(* IEC 61131-3 sources: plc_simulator/services/codesys/POUs (part 3) *)

(* ---- FC_TSK_Resolve.st ---- *)
(* ===========================================================================================
 *  FC_TSK_Resolve — Conflict resolution
 *
 *  Company : Galvatek part of the John Cockerill Group
 *  Author  : Jarmo Piipponen
 *  Created : 25.03.2026
 *
 * -------------------------------------------------------------------------------------------
 *  Four sequential resolution phases:
 *  1. ADVANCE (chain bottleneck + suffix flex_down)
 *  2. DELAY (single-stage vFlexUp)
 *  3. PRECEDING_DELAY (conf stage-1)
 *  4. DELAY_PREV_PAST_NEXT (force order swap)
 *
 *  VAR_IN_OUT: ioSchedule, ioTask, ioBatch, ioLocks,
 *  ioLockCnt — caller passes live or workspace arrays.
 *
 *  ------------------------------------------------------------------------------------------
 *
 *  Changes:
 *
 *
 *
 *)

FUNCTION FC_TSK_Resolve : BOOL

(* Introduction of Variables ----------------------------------------------------------------*)

VAR_INPUT
  iConfUnit               : INT;
  iConfStage              : INT;
  iConfTrans              : INT;
  iBlockedUnit            : INT;
  iBlockedStage           : INT;
  iDeficit                 : REAL;
END_VAR

VAR_IN_OUT  (* array sizes must match GVL_JC_Constants: 50=MAX_LOCKS, 10=MAX_UNITS, 3=MAX_TRANSPORTERS *)
  ioLocks                  : ARRAY[1..50] OF UDT_JC_TskLockType;
  ioLockCnt               : INT;
  ioSchedule               : ARRAY[1..10] OF UDT_JC_TskScheduleType;
  ioTask                   : ARRAY[1..3] OF UDT_JC_TskQueueType;
  ioBatch                  : ARRAY[1..10] OF UDT_BatchType;
END_VAR

VAR_EXTERNAL CONSTANT
    MAX_TRANSPORTERS        : INT;
    MAX_UNITS               : INT;
    SCH_TSK_FLEX_FACTOR     : REAL;
END_VAR

VAR_OUTPUT
  oSolved                  : BOOL;
  oTotalDelay             : REAL;
  oTotalAdv               : REAL;
END_VAR

VAR
  vRemain                    : REAL;
  cap                       : REAL;
  vAmount                    : REAL;
  vStageFlex                : REAL;
  is_locked_adv             : BOOL;
  is_locked_del             : BOOL;
  vCanAdvance               : BOOL;
  vCanDelay                 : BOOL;
  vLockI                    : INT;
  vPrevConfStage           : INT;
  is_pcs_locked             : BOOL;
  vPrevSinkStn             : INT;
  vNextLiftStn             : INT;
  is_blk_adv_locked         : BOOL;
  qi                        : INT;
  vChainFlex                : REAL;
  vSuffixFlex               : REAL;
  earlier_stg               : INT;
  earlier_flex              : REAL;
  vChainAmount              : REAL;
  vSuffixAmount             : REAL;
  vSchedBlocked             : INT;
  vSchedConf                : INT;
  vSchedPrevConf           : INT;
  vTmpSi                    : INT;
  cap_remain                : REAL;
END_VAR

FC_TSK_Resolve := FALSE;
oSolved      := FALSE;
oTotalDelay := 0.0;
oTotalAdv   := 0.0;
vRemain        := iDeficit;

IF vRemain <= 0.1 THEN
  oSolved := TRUE;
  FC_TSK_Resolve := TRUE;
  RETURN;
END_IF;

(* Lock check: blocked stage locked DELAY? cannot ADVANCE *)
is_locked_adv := FALSE;
FOR vLockI := 1 TO ioLockCnt DO
  IF ioLocks[vLockI].Unit = iBlockedUnit
     AND ioLocks[vLockI].Stage = iBlockedStage
     AND ioLocks[vLockI].Direction = 2 THEN
    is_locked_adv := TRUE;
  END_IF;
END_FOR;

(* Lock check: conf stage locked ADVANCE? cannot DELAY *)
is_locked_del := FALSE;
FOR vLockI := 1 TO ioLockCnt DO
  IF ioLocks[vLockI].Unit = iConfUnit
     AND ioLocks[vLockI].Stage = iConfStage
     AND ioLocks[vLockI].Direction = 1 THEN
    is_locked_del := TRUE;
  END_IF;
END_FOR;

vCanAdvance := NOT is_locked_adv;
vCanDelay   := NOT is_locked_del;

(* Map ProgramStage to schedule array index *)
vSchedBlocked := 0;
IF iBlockedUnit >= 1 AND iBlockedUnit <= MAX_UNITS THEN
  FOR vTmpSi := 1 TO ioSchedule[iBlockedUnit].StageCount DO
    IF ioSchedule[iBlockedUnit].Stages[vTmpSi].ProgramStage = iBlockedStage THEN
      vSchedBlocked := vTmpSi; EXIT;
    END_IF;
  END_FOR;
END_IF;

vSchedConf := 0;
IF iConfUnit >= 1 AND iConfUnit <= MAX_UNITS THEN
  FOR vTmpSi := 1 TO ioSchedule[iConfUnit].StageCount DO
    IF ioSchedule[iConfUnit].Stages[vTmpSi].ProgramStage = iConfStage THEN
      vSchedConf := vTmpSi; EXIT;
    END_IF;
  END_FOR;
END_IF;

(* ================================================================ *)
(* PHASE 1: ADVANCE -- advance blocked batch                       *)
(* ================================================================ *)
IF vCanAdvance
   AND iBlockedUnit >= 1 AND iBlockedUnit <= MAX_UNITS
   AND iBlockedStage >= 1 THEN
IF vSchedBlocked >= 1 AND vSchedBlocked <= ioSchedule[iBlockedUnit].StageCount THEN

  (* Absolute flex cap: use (MaxTime - MinTime) range, not (CalcTime - MinTime).
     This prevents cumulative drift when CalcTime is vAdjusted across rounds. *)
  vStageFlex := DINT_TO_REAL(
    ioSchedule[iBlockedUnit].Stages[vSchedBlocked].MaxTime
    - ioSchedule[iBlockedUnit].Stages[vSchedBlocked].MinTime);
  IF vStageFlex < 0.0 THEN vStageFlex := 0.0; END_IF;
  vStageFlex := vStageFlex * SCH_TSK_FLEX_FACTOR;
  (* Cap to actual remaining advance room *)
  cap_remain := DINT_TO_REAL(
    ioSchedule[iBlockedUnit].Stages[vSchedBlocked].CalcTime
    - ioSchedule[iBlockedUnit].Stages[vSchedBlocked].MinTime);
  IF cap_remain < 0.0 THEN cap_remain := 0.0; END_IF;
  IF vStageFlex > cap_remain THEN vStageFlex := cap_remain; END_IF;

  IF vStageFlex > 0.1 THEN
    IF ioBatch[iBlockedUnit].CurStage = iBlockedStage THEN cap := 0.9;
  ELSE cap := 0.5; END_IF;

    (* Chain bottleneck search *)
    vChainFlex := vStageFlex;
    FOR earlier_stg := 1 TO vSchedBlocked - 1 DO
      earlier_flex := DINT_TO_REAL(
        ioSchedule[iBlockedUnit].Stages[earlier_stg].CalcTime
        - ioSchedule[iBlockedUnit].Stages[earlier_stg].MinTime);
  IF earlier_flex < 0.0 THEN earlier_flex := 0.0; END_IF;
      IF earlier_flex > 0.0 AND earlier_flex < vChainFlex THEN
        vChainFlex := earlier_flex;
      END_IF;
    END_FOR;

    (* CHAIN_ADVANCE *)
    vChainAmount := vChainFlex * cap;
  IF vChainAmount > vRemain THEN vChainAmount := vRemain; END_IF;

    IF vChainAmount > 0.1 THEN
      ioSchedule[iBlockedUnit].Stages[vSchedBlocked].CalcTime :=
        ioSchedule[iBlockedUnit].Stages[vSchedBlocked].CalcTime - REAL_TO_DINT(vChainAmount);
      ioSchedule[iBlockedUnit].Stages[vSchedBlocked].ExitTime :=
        ioSchedule[iBlockedUnit].Stages[vSchedBlocked].ExitTime - REAL_TO_LINT(vChainAmount);

      FC_STC_ShiftSchedule(iUnit := iBlockedUnit, iFromStage := iBlockedStage + 1,
                         iAmount := -vChainAmount, ioSchedule := ioSchedule, ioTask := ioTask);

      ioBatch[iBlockedUnit].CalTime :=
        ioBatch[iBlockedUnit].CalTime - REAL_TO_DINT(vChainAmount);
      IF ioBatch[iBlockedUnit].CalTime < ioBatch[iBlockedUnit].MinTime THEN
        ioBatch[iBlockedUnit].CalTime := ioBatch[iBlockedUnit].MinTime;
      END_IF;

      vRemain := vRemain - vChainAmount;
      oTotalAdv := oTotalAdv + vChainAmount;
    END_IF;

    (* SUFFIX_ADVANCE *)
    vSuffixFlex := vStageFlex - vChainFlex;
    IF vSuffixFlex > 0.1 AND vRemain > 0.1 THEN
      vSuffixAmount := vSuffixFlex * cap;
  IF vSuffixAmount > vRemain THEN vSuffixAmount := vRemain; END_IF;

      IF vSuffixAmount > 0.1 THEN
        ioSchedule[iBlockedUnit].Stages[vSchedBlocked].CalcTime :=
          ioSchedule[iBlockedUnit].Stages[vSchedBlocked].CalcTime - REAL_TO_DINT(vSuffixAmount);
        ioSchedule[iBlockedUnit].Stages[vSchedBlocked].ExitTime :=
          ioSchedule[iBlockedUnit].Stages[vSchedBlocked].ExitTime - REAL_TO_LINT(vSuffixAmount);

        FC_STC_ShiftSchedule(iUnit := iBlockedUnit, iFromStage := iBlockedStage + 1,
                           iAmount := -vSuffixAmount, ioSchedule := ioSchedule, ioTask := ioTask);

        ioBatch[iBlockedUnit].CalTime :=
          ioBatch[iBlockedUnit].CalTime - REAL_TO_DINT(vSuffixAmount);
        IF ioBatch[iBlockedUnit].CalTime < ioBatch[iBlockedUnit].MinTime THEN
          ioBatch[iBlockedUnit].CalTime := ioBatch[iBlockedUnit].MinTime;
        END_IF;

        vRemain := vRemain - vSuffixAmount;
        oTotalAdv := oTotalAdv + vSuffixAmount;
      END_IF;
    END_IF;

    (* Record lock: ADVANCE on blocked stage *)
    IF ioLockCnt < 50 THEN
      ioLockCnt := ioLockCnt + 1;
      ioLocks[ioLockCnt].Unit := iBlockedUnit;
      ioLocks[ioLockCnt].Stage := iBlockedStage;
      ioLocks[ioLockCnt].Direction := 1;
    END_IF;

    IF vRemain <= 0.1 THEN
  oSolved := TRUE;
  FC_TSK_Resolve := TRUE; RETURN;
    END_IF;
  END_IF;
END_IF;
END_IF;

(* ================================================================ *)
(* PHASE 2: DELAY -- vDelay vConflict batch                          *)
(* ================================================================ *)
IF vCanDelay AND vRemain > 0.1
   AND iConfUnit >= 1 AND iConfUnit <= MAX_UNITS
   AND iConfStage >= 1 THEN
IF vSchedConf >= 1 AND vSchedConf <= ioSchedule[iConfUnit].StageCount THEN

  (* Absolute flex cap: use (MaxTime - MinTime) range, not (MaxTime - CalcTime).
     This prevents cumulative drift when CalcTime is vAdjusted across rounds. *)
  vStageFlex := DINT_TO_REAL(
    ioSchedule[iConfUnit].Stages[vSchedConf].MaxTime
    - ioSchedule[iConfUnit].Stages[vSchedConf].MinTime);
  IF vStageFlex < 0.0 THEN vStageFlex := 0.0; END_IF;
  vStageFlex := vStageFlex * SCH_TSK_FLEX_FACTOR;
  (* Cap to actual remaining vDelay room *)
  cap_remain := DINT_TO_REAL(
    ioSchedule[iConfUnit].Stages[vSchedConf].MaxTime
    - ioSchedule[iConfUnit].Stages[vSchedConf].CalcTime);
  IF cap_remain < 0.0 THEN cap_remain := 0.0; END_IF;
  IF vStageFlex > cap_remain THEN vStageFlex := cap_remain; END_IF;

  IF vStageFlex > 0.1 THEN
    IF ioBatch[iConfUnit].CurStage = iConfStage THEN cap := 0.9;
  ELSE cap := 0.5; END_IF;
    vAmount := vStageFlex * cap;
  IF vAmount > vRemain THEN vAmount := vRemain; END_IF;

    ioSchedule[iConfUnit].Stages[vSchedConf].CalcTime :=
      ioSchedule[iConfUnit].Stages[vSchedConf].CalcTime + REAL_TO_DINT(vAmount);
    ioSchedule[iConfUnit].Stages[vSchedConf].ExitTime :=
      ioSchedule[iConfUnit].Stages[vSchedConf].ExitTime + REAL_TO_LINT(vAmount);

    FC_STC_ShiftSchedule(iUnit := iConfUnit, iFromStage := iConfStage + 1,
                       iAmount := vAmount, ioSchedule := ioSchedule, ioTask := ioTask);

    IF ioBatch[iConfUnit].CurStage = iConfStage THEN
      ioBatch[iConfUnit].CalTime :=
        ioBatch[iConfUnit].CalTime + REAL_TO_DINT(vAmount);
      IF ioBatch[iConfUnit].CalTime > ioBatch[iConfUnit].MaxTime THEN
        ioBatch[iConfUnit].CalTime := ioBatch[iConfUnit].MaxTime;
      END_IF;
    END_IF;

    vRemain := vRemain - vAmount;
    oTotalDelay := oTotalDelay + vAmount;

    IF ioLockCnt < 50 THEN
      ioLockCnt := ioLockCnt + 1;
      ioLocks[ioLockCnt].Unit := iConfUnit;
      ioLocks[ioLockCnt].Stage := iConfStage;
      ioLocks[ioLockCnt].Direction := 2;
    END_IF;

    IF vRemain <= 0.1 THEN
  oSolved := TRUE;
  FC_TSK_Resolve := TRUE; RETURN;
    END_IF;
  END_IF;
END_IF;
END_IF;

(* ================================================================ *)
(* PHASE 3: PRECEDING_DELAY -- vDelay conf batch at stage-1         *)
(* ================================================================ *)
vPrevConfStage := iConfStage - 1;

vSchedPrevConf := 0;
IF iConfUnit >= 1 AND iConfUnit <= MAX_UNITS AND vPrevConfStage >= 1 THEN
  FOR vTmpSi := 1 TO ioSchedule[iConfUnit].StageCount DO
    IF ioSchedule[iConfUnit].Stages[vTmpSi].ProgramStage = vPrevConfStage THEN
  vSchedPrevConf := vTmpSi; EXIT;
    END_IF;
  END_FOR;
END_IF;

IF vRemain > 0.1 AND vPrevConfStage >= 1 AND iConfUnit >= 1 AND iConfUnit <= MAX_UNITS
   AND vSchedPrevConf >= 1 THEN
  is_pcs_locked := FALSE;
  FOR vLockI := 1 TO ioLockCnt DO
    IF ioLocks[vLockI].Unit = iConfUnit
       AND ioLocks[vLockI].Stage = vPrevConfStage
       AND ioLocks[vLockI].Direction = 1 THEN
      is_pcs_locked := TRUE;
    END_IF;
  END_FOR;

  IF NOT is_pcs_locked THEN
    (* Flex cap: min + factor × (max - min); available room = vFlexCap - CalcTime *)
    vStageFlex := DINT_TO_REAL(
      ioSchedule[iConfUnit].Stages[vSchedPrevConf].MinTime
      + REAL_TO_DINT(SCH_TSK_FLEX_FACTOR * DINT_TO_REAL(
          ioSchedule[iConfUnit].Stages[vSchedPrevConf].MaxTime
        - ioSchedule[iConfUnit].Stages[vSchedPrevConf].MinTime))
      - ioSchedule[iConfUnit].Stages[vSchedPrevConf].CalcTime);
  IF vStageFlex < 0.0 THEN vStageFlex := 0.0; END_IF;

    IF vStageFlex > 0.1 THEN
      IF ioBatch[iConfUnit].CurStage = vPrevConfStage THEN cap := 0.9;
  ELSE cap := 0.5; END_IF;
      vAmount := vStageFlex * cap;
  IF vAmount > vRemain THEN vAmount := vRemain; END_IF;

      ioSchedule[iConfUnit].Stages[vSchedPrevConf].CalcTime :=
        ioSchedule[iConfUnit].Stages[vSchedPrevConf].CalcTime + REAL_TO_DINT(vAmount);
      ioSchedule[iConfUnit].Stages[vSchedPrevConf].ExitTime :=
        ioSchedule[iConfUnit].Stages[vSchedPrevConf].ExitTime + REAL_TO_LINT(vAmount);
      FC_STC_ShiftSchedule(iUnit := iConfUnit, iFromStage := vPrevConfStage + 1,
                         iAmount := vAmount, ioSchedule := ioSchedule, ioTask := ioTask);

      IF ioBatch[iConfUnit].CurStage = iConfStage THEN
        ioBatch[iConfUnit].CalTime :=
          ioBatch[iConfUnit].CalTime + REAL_TO_DINT(vAmount);
        IF ioBatch[iConfUnit].CalTime > ioBatch[iConfUnit].MaxTime THEN
          ioBatch[iConfUnit].CalTime := ioBatch[iConfUnit].MaxTime;
        END_IF;
      END_IF;

      vRemain := vRemain - vAmount;
      oTotalDelay := oTotalDelay + vAmount;

      IF ioLockCnt < 50 THEN
        ioLockCnt := ioLockCnt + 1;
        ioLocks[ioLockCnt].Unit := iConfUnit;
        ioLocks[ioLockCnt].Stage := vPrevConfStage;
        ioLocks[ioLockCnt].Direction := 2;
      END_IF;

      IF vRemain <= 0.1 THEN
  oSolved := TRUE;
  FC_TSK_Resolve := TRUE; RETURN;
      END_IF;
    END_IF;
  END_IF;
END_IF;

(* ================================================================ *)
(* PHASE 4: DELAY_PREV_PAST_NEXT -- force order swap               *)
(* ================================================================ *)
IF vRemain > 0.1 AND iBlockedUnit >= 1 AND iBlockedUnit <= MAX_UNITS THEN
  vPrevSinkStn := 0;
  vNextLiftStn := 0;
  IF iConfTrans >= 1 AND iConfTrans <= MAX_TRANSPORTERS THEN
    FOR qi := 1 TO ioTask[iConfTrans].Count DO
      IF ioTask[iConfTrans].Queue[qi].Unit = iBlockedUnit
         AND ioTask[iConfTrans].Queue[qi].Stage = iBlockedStage THEN
        vPrevSinkStn := ioTask[iConfTrans].Queue[qi].SinkStationTarget;
      END_IF;
      IF ioTask[iConfTrans].Queue[qi].Unit = iConfUnit
         AND ioTask[iConfTrans].Queue[qi].Stage = iConfStage THEN
        vNextLiftStn := ioTask[iConfTrans].Queue[qi].LiftStationTarget;
      END_IF;
    END_FOR;
  END_IF;

  IF NOT (vPrevSinkStn > 0 AND vNextLiftStn > 0 AND vPrevSinkStn = vNextLiftStn) THEN
    is_blk_adv_locked := FALSE;
    FOR vLockI := 1 TO ioLockCnt DO
      IF ioLocks[vLockI].Unit = iBlockedUnit
         AND ioLocks[vLockI].Stage = iBlockedStage
         AND ioLocks[vLockI].Direction = 1 THEN
        is_blk_adv_locked := TRUE;
      END_IF;
    END_FOR;

    IF NOT is_blk_adv_locked THEN
      (* Flex cap: min + factor × (max - min); available room = vFlexCap - CalcTime *)
      vStageFlex := DINT_TO_REAL(
        ioSchedule[iBlockedUnit].Stages[vSchedBlocked].MinTime
        + REAL_TO_DINT(SCH_TSK_FLEX_FACTOR * DINT_TO_REAL(
            ioSchedule[iBlockedUnit].Stages[vSchedBlocked].MaxTime
          - ioSchedule[iBlockedUnit].Stages[vSchedBlocked].MinTime))
        - ioSchedule[iBlockedUnit].Stages[vSchedBlocked].CalcTime);
  IF vStageFlex < 0.0 THEN vStageFlex := 0.0; END_IF;

      IF vStageFlex > 0.1 THEN
        IF ioBatch[iBlockedUnit].CurStage = iBlockedStage THEN cap := 0.9;
  ELSE cap := 0.5; END_IF;
        vAmount := vStageFlex * cap;
  IF vAmount > vRemain THEN vAmount := vRemain; END_IF;

        ioSchedule[iBlockedUnit].Stages[vSchedBlocked].CalcTime :=
          ioSchedule[iBlockedUnit].Stages[vSchedBlocked].CalcTime + REAL_TO_DINT(vAmount);
        ioSchedule[iBlockedUnit].Stages[vSchedBlocked].ExitTime :=
          ioSchedule[iBlockedUnit].Stages[vSchedBlocked].ExitTime + REAL_TO_LINT(vAmount);
        FC_STC_ShiftSchedule(iUnit := iBlockedUnit, iFromStage := iBlockedStage + 1,
                           iAmount := vAmount, ioSchedule := ioSchedule, ioTask := ioTask);

        IF ioBatch[iBlockedUnit].CurStage = iBlockedStage THEN
          ioBatch[iBlockedUnit].CalTime :=
            ioBatch[iBlockedUnit].CalTime + REAL_TO_DINT(vAmount);
          IF ioBatch[iBlockedUnit].CalTime > ioBatch[iBlockedUnit].MaxTime THEN
            ioBatch[iBlockedUnit].CalTime := ioBatch[iBlockedUnit].MaxTime;
          END_IF;
        END_IF;

        vRemain := vRemain - vAmount;
        oTotalDelay := oTotalDelay + vAmount;

        IF ioLockCnt < 50 THEN
          ioLockCnt := ioLockCnt + 1;
          ioLocks[ioLockCnt].Unit := iBlockedUnit;
          ioLocks[ioLockCnt].Stage := iBlockedStage;
          ioLocks[ioLockCnt].Direction := 2;
        END_IF;

        IF vRemain <= 0.1 THEN
  oSolved := TRUE;
  FC_TSK_Resolve := TRUE; RETURN;
        END_IF;
      END_IF;
    END_IF;
  END_IF;
END_IF;

END_FUNCTION

(* ---- STC_CalcHorizontalTravel.st ---- *)
(* ===========================================================================================
 *  STC_CalcHorizontalTravel — Horizontal travel time
 *
 *  Company : Galvatek part of the John Cockerill Group
 *  Author  : Jarmo Piipponen
 *  Created : 25.03.2026
 *
 * -------------------------------------------------------------------------------------------
 *  Calculates horizontal travel time between two stations
 *  (no lift/sink) using precomputed move time table.
 *  Caller passes i_move (UDT_JC_MoveTimesType) for the
 *  specific transporter.
 *
 *  ------------------------------------------------------------------------------------------
 *
 *  Changes:
 *
 *
 *
 *)

FUNCTION STC_CalcHorizontalTravel : REAL

(* Introduction of Variables ----------------------------------------------------------------*)

VAR_INPUT
  i_from_stn                : INT;     (* source station number *)
  i_to_stn                  : INT;     (* destination station number *)
  i_move                    : UDT_JC_MoveTimesType;   (* transporter's precomputed move times *)
END_VAR

VAR
  from_idx                  : INT;
  to_idx                    : INT;
END_VAR

STC_CalcHorizontalTravel := 0.0;
IF i_from_stn > 0 AND i_to_stn > 0 AND i_from_stn <> i_to_stn THEN
  from_idx := i_from_stn - MIN_STATION_INDEX;
  to_idx   := i_to_stn - MIN_STATION_INDEX;
  IF from_idx >= 1 AND from_idx <= 25 AND to_idx >= 1 AND to_idx <= 25 THEN
    STC_CalcHorizontalTravel := INT_TO_REAL(i_move.Travel[from_idx].ToTime[to_idx]) / 10.0;
  END_IF;
END_IF;

END_FUNCTION

(* ---- STC_CalcSchedule.st ---- *)
(* ===========================================================================================
 *  STC_CalcSchedule — Calculate batch schedule for one unit
 *
 *  Company : Galvatek part of the John Cockerill Group
 *  Author  : Jarmo Piipponen
 *  Created : 25.03.2026
 *
 * -------------------------------------------------------------------------------------------
 *  Shared FC: both TSK and DEP call this with different arrays.
 *  Calculates start/finish times for each treatment stage based
 *  on elapsed time, cal_time and transfer durations.
 *
 *  ------------------------------------------------------------------------------------------
 *
 *  Changes:
 *
 *
 *
 *)

FUNCTION STC_CalcSchedule : BOOL

(* Introduction of Variables ----------------------------------------------------------------*)

VAR_INPUT
  i_unit                    : INT;
  i_trans                   : INT;
  i_time_s                  : LINT;
END_VAR

VAR_IN_OUT  (* array sizes must match GVL_JC_Constants: 10=MAX_UNITS *)
  io_schedule               : ARRAY[1..10] OF UDT_JC_TskScheduleType;
  io_batch                  : ARRAY[1..10] OF UDT_BatchType;
  io_program                : ARRAY[1..10] OF UDT_TreatmentProgramType;
END_VAR

VAR_EXTERNAL CONSTANT
    MIN_STATION_INDEX        : INT;
    MAX_STATION_INDEX        : INT;
    MAX_UNITS               : INT;
    MAX_TRANSPORTERS        : INT;
    MAX_STEPS_PER_PROGRAM   : INT;
    NOT_PROCESSED           : INT;
    USED                    : INT;
END_VAR

VAR_EXTERNAL
  g_unit                    : ARRAY[1..MAX_UNITS] OF UDT_JC_UnitType;
  Stations                 : ARRAY[MIN_STATION_INDEX..MAX_STATION_INDEX] OF UDT_StationType;
  g_station_occupancy             : ARRAY[1..MAX_STATION_INDEX] OF UDT_JC_UnitAtStationType;
  CountStations              : INT;
  g_move                    : ARRAY[1..MAX_TRANSPORTERS] OF UDT_JC_MoveTimesType;
  Transporters                     : ARRAY[0..MAX_TRANSPORTERS] OF UDT_TransporterType;
  g_transporter             : ARRAY[1..MAX_TRANSPORTERS] OF UDT_TransporterStatusType;
END_VAR

VAR
  stg                       : INT;
  stn_num                   : INT;
  prev_stn                  : INT;
  cur_stage                 : INT;
  location                  : INT;
  start_st                  : INT;
  entry_t                   : LINT;
  exit_t                    : LINT;
  xfer_t                    : REAL;
  calc_s                    : REAL;
  min_s                     : REAL;
  max_s                     : REAL;
  is_on_stn                 : BOOL;
  is_first                  : BOOL;
  remain_s                  : REAL;
  elapsed_s                 : REAL;
  p                         : INT;
  chosen_stn                : INT;
  tmp_move                  : UDT_JC_MoveTimesType;
  cand_arr                  : ARRAY[1..5] OF INT;
  cand_cnt                  : INT;
  sched_occupied            : ARRAY[1..5] OF BOOL;
  best_change_time          : LINT;
  my_entry                  : LINT;
  my_exit                   : LINT;
  ov_start                  : LINT;
  ov_end                    : LINT;
  uj                        : INT;
  sj                        : INT;
END_VAR

STC_CalcSchedule := FALSE;
IF i_unit < 1 OR i_unit > MAX_UNITS THEN RETURN; END_IF;
IF i_trans < 1 OR i_trans > MAX_TRANSPORTERS THEN RETURN; END_IF;

cur_stage := io_batch[i_unit].CurStage;
location  := g_unit[i_unit].location;
is_on_stn := location >= MIN_STATION_INDEX;

(* Clear old schedule *)
FOR stg := 0 TO MAX_STEPS_PER_PROGRAM DO
  io_schedule[i_unit].Stages[stg].station := 0;
  io_schedule[i_unit].Stages[stg].ProgramStage := 0;
  io_schedule[i_unit].Stages[stg].EntryTime := 0;
  io_schedule[i_unit].Stages[stg].ExitTime := 0;
  io_schedule[i_unit].Stages[stg].MinTime := 0;
  io_schedule[i_unit].Stages[stg].CalcTime := 0;
  io_schedule[i_unit].Stages[stg].MaxTime := 0;
  io_schedule[i_unit].Stages[stg].TransferTime := 0;
END_FOR;
io_schedule[i_unit].StageCount := 0;

(* Waiting batch (state = NOT_PROCESSED): treat as stage 0 *)
IF io_batch[i_unit].State = NOT_PROCESSED THEN
  cur_stage := 0;
END_IF;

IF is_on_stn THEN
  start_st := cur_stage;
ELSE
  start_st := cur_stage + 1;
END_IF;
IF start_st < 1 THEN
  start_st := 1;
END_IF;

IF is_on_stn THEN
  prev_stn := location;
ELSIF cur_stage >= 1 AND cur_stage <= 30 THEN
  prev_stn := io_program[i_unit].Steps[cur_stage].Stations[0];
ELSE
  prev_stn := 0;
END_IF;

exit_t := i_time_s;
is_first := TRUE;

(* Prepend current location to Stages[0] when unit needs pre-positioning *)
IF is_on_stn AND start_st >= 1 THEN
  stn_num := 0;
  FOR p := 0 TO 4 DO
    IF io_program[i_unit].Steps[start_st].Stations[p] = location THEN
      stn_num := location;
    END_IF;
  END_FOR;
  IF stn_num = 0 THEN
    io_schedule[i_unit].Stages[0].station       := location;
    io_schedule[i_unit].Stages[0].ProgramStage := 0;
    io_schedule[i_unit].Stages[0].EntryTime    := exit_t;
    io_schedule[i_unit].Stages[0].TransferTime := 0;

    IF io_batch[i_unit].CurStage = 0 AND io_batch[i_unit].CalTime > 0 THEN
      IF io_batch[i_unit].StartTime > 0 AND io_batch[i_unit].StartTime < i_time_s THEN
        elapsed_s := LINT_TO_REAL(i_time_s - io_batch[i_unit].StartTime);
      ELSE
        elapsed_s := 0.0;
      END_IF;
      remain_s := DINT_TO_REAL(io_batch[i_unit].CalTime) - elapsed_s;
  IF remain_s < 1.0 THEN remain_s := 1.0; END_IF;
      exit_t := i_time_s + REAL_TO_LINT(remain_s);
      io_schedule[i_unit].Stages[0].ExitTime  := exit_t;
      io_schedule[i_unit].Stages[0].CalcTime  := REAL_TO_DINT(remain_s);
      io_schedule[i_unit].Stages[0].MinTime   := io_batch[i_unit].MinTime;
      io_schedule[i_unit].Stages[0].MaxTime   := io_batch[i_unit].MaxTime;
    ELSE
      (* Pickup wait: transporter horizontal travel time to this station, min 5s *)
      calc_s := STC_CalcHorizontalTravel(
        i_from_stn := g_transporter[i_trans].CurrentStation,
        i_to_stn   := location,
        i_move     := g_move[i_trans]);
      IF calc_s < 5.0 THEN calc_s := 5.0; END_IF;
      exit_t := i_time_s + REAL_TO_LINT(calc_s);
      io_schedule[i_unit].Stages[0].ExitTime  := exit_t;
      io_schedule[i_unit].Stages[0].CalcTime  := REAL_TO_DINT(calc_s);
      io_schedule[i_unit].Stages[0].MinTime   := REAL_TO_DINT(calc_s);
      io_schedule[i_unit].Stages[0].MaxTime   := REAL_TO_DINT(2.0 * calc_s);
    END_IF;

    is_first := FALSE;
  END_IF;
END_IF;

(* ============================================================
   MAIN LOOP: Calculate schedule for each program stage
   ============================================================ *)
FOR stg := start_st TO io_program[i_unit].StepCount DO

  cand_cnt := 0;
  FOR p := 0 TO 4 DO
    IF io_program[i_unit].Steps[stg].Stations[p] > 0 THEN
      cand_cnt := cand_cnt + 1;
      cand_arr[cand_cnt] := io_program[i_unit].Steps[stg].Stations[p];
      sched_occupied[cand_cnt] := FALSE;
    END_IF;
  END_FOR;

  IF cand_cnt = 0 THEN
    EXIT;
  END_IF;

  chosen_stn := 0;
  IF is_first AND is_on_stn AND stg = cur_stage THEN
    FOR p := 1 TO cand_cnt DO
      IF cand_arr[p] = location THEN
        chosen_stn := location;
      END_IF;
    END_FOR;
  END_IF;

  IF chosen_stn = 0 THEN
    IF cand_cnt = 1 THEN
      chosen_stn := cand_arr[1];
    ELSE
      (* Estimate this batch's time window per candidate for overlap check *)
      calc_s := DINT_TO_REAL(io_program[i_unit].Steps[stg].CalTime);
      tmp_move := g_move[i_trans];

      FOR p := 1 TO cand_cnt DO
        (* Calculate entry/exit per candidate station individually *)
        xfer_t := STC_CalcTransferTime(
          i_from_stn            := prev_stn,
          i_to_stn              := cand_arr[p],
          i_move                := tmp_move,
          i_from_dropping_x10   := Stations[prev_stn].DrippingTime,
          i_to_device_delay_x10 := Stations[cand_arr[p]].DeviceDelay,
          i_drip_tray_delay_x10 := Transporters[i_trans].DripTrayDelay
        );
        my_entry := exit_t + REAL_TO_LINT(xfer_t);
        my_exit  := my_entry + REAL_TO_LINT(calc_s);

        FOR uj := 1 TO MAX_UNITS DO
          IF uj <> i_unit AND io_schedule[uj].StageCount > 0 THEN
            FOR sj := 0 TO io_schedule[uj].StageCount DO
              IF io_schedule[uj].Stages[sj].station = cand_arr[p] THEN
                ov_start := my_entry;
                IF io_schedule[uj].Stages[sj].EntryTime > ov_start THEN
                  ov_start := io_schedule[uj].Stages[sj].EntryTime;
                END_IF;
                ov_end := my_exit;
                IF io_schedule[uj].Stages[sj].ExitTime < ov_end THEN
                  ov_end := io_schedule[uj].Stages[sj].ExitTime;
                END_IF;
                IF ov_end > ov_start THEN
                  sched_occupied[p] := TRUE;
                END_IF;
              END_IF;
            END_FOR;
          END_IF;
        END_FOR;

      END_FOR;

      (* Pass 1: prefer schedule-free station, pick earliest ChangeTime *)
      best_change_time := LINT#9999999999;
      FOR p := 1 TO cand_cnt DO
        IF NOT sched_occupied[p] THEN
          IF cand_arr[p] >= MIN_STATION_INDEX AND cand_arr[p] <= MAX_STATION_INDEX THEN
            IF g_station_occupancy[cand_arr[p]].ChangeTime < best_change_time THEN
              best_change_time := g_station_occupancy[cand_arr[p]].ChangeTime;
              chosen_stn := cand_arr[p];
            END_IF;
          END_IF;
        END_IF;
      END_FOR;

      (* Pass 2: all sched-occupied — pick first candidate *)
      IF chosen_stn = 0 THEN
        chosen_stn := cand_arr[1];
      END_IF;
    END_IF;
  END_IF;

  stn_num := chosen_stn;

  calc_s := DINT_TO_REAL(io_program[i_unit].Steps[stg].CalTime);
  min_s  := DINT_TO_REAL(io_program[i_unit].Steps[stg].MinTime);
  max_s  := DINT_TO_REAL(io_program[i_unit].Steps[stg].MaxTime);

  tmp_move := g_move[i_trans];
  IF prev_stn >= MIN_STATION_INDEX AND prev_stn <= MAX_STATION_INDEX
     AND stn_num >= MIN_STATION_INDEX AND stn_num <= MAX_STATION_INDEX THEN
    IF Stations[prev_stn].Crosstransport > 0
       AND Stations[prev_stn].ChangeStation > 0
       AND Stations[prev_stn].YPosition <> Stations[stn_num].YPosition THEN
      xfer_t := INT_TO_REAL(Stations[prev_stn].CrossTransportTime)
              + STC_CalcTransferTime(
                  i_from_stn            := Stations[prev_stn].ChangeStation,
                  i_to_stn              := stn_num,
                  i_move                := tmp_move,
                  i_from_dropping_x10   := Stations[Stations[prev_stn].ChangeStation].DrippingTime,
                  i_to_device_delay_x10 := Stations[stn_num].DeviceDelay,
                  i_drip_tray_delay_x10 := Transporters[i_trans].DripTrayDelay
                );
    ELSE
      xfer_t := STC_CalcTransferTime(
        i_from_stn            := prev_stn,
        i_to_stn              := stn_num,
        i_move                := tmp_move,
        i_from_dropping_x10   := Stations[prev_stn].DrippingTime,
        i_to_device_delay_x10 := Stations[stn_num].DeviceDelay,
        i_drip_tray_delay_x10 := Transporters[i_trans].DripTrayDelay
      );
    END_IF;
  ELSE
    xfer_t := 60.0;
  END_IF;

  IF is_first AND is_on_stn AND stg = cur_stage THEN
    entry_t := i_time_s;
    IF io_batch[i_unit].StartTime > 0 THEN
      elapsed_s := LINT_TO_REAL(i_time_s - io_batch[i_unit].StartTime);
    ELSE
      elapsed_s := 0.0;
    END_IF;
    remain_s := DINT_TO_REAL(io_batch[i_unit].CalTime) - elapsed_s;
  IF remain_s < 1.0 THEN remain_s := 1.0; END_IF;
    exit_t := i_time_s + REAL_TO_LINT(remain_s);
  ELSIF is_first AND NOT is_on_stn THEN
    IF io_batch[i_unit].StartTime > 0 AND io_batch[i_unit].CalTime > 0 THEN
      entry_t := io_batch[i_unit].StartTime + DINT_TO_LINT(io_batch[i_unit].CalTime);
    ELSE
      entry_t := i_time_s + REAL_TO_LINT(xfer_t);
    END_IF;
    exit_t  := entry_t + REAL_TO_LINT(calc_s);
  ELSE
    entry_t := exit_t + REAL_TO_LINT(xfer_t);
    exit_t  := entry_t + REAL_TO_LINT(calc_s);
  END_IF;

  IF stg <= 30 THEN
    io_schedule[i_unit].Stages[stg].station       := stn_num;
    io_schedule[i_unit].Stages[stg].ProgramStage := stg;
    io_schedule[i_unit].Stages[stg].EntryTime    := entry_t;
    io_schedule[i_unit].Stages[stg].ExitTime     := exit_t;
    io_schedule[i_unit].Stages[stg].MinTime      := REAL_TO_DINT(min_s);
    io_schedule[i_unit].Stages[stg].CalcTime     := REAL_TO_DINT(calc_s);
    io_schedule[i_unit].Stages[stg].MaxTime      := REAL_TO_DINT(max_s);
    io_schedule[i_unit].Stages[stg].TransferTime := REAL_TO_DINT(xfer_t);
    io_schedule[i_unit].StageCount := stg;
  END_IF;

  prev_stn := stn_num;
  is_first := FALSE;

END_FOR;

STC_CalcSchedule := TRUE;

END_FUNCTION

(* ---- STC_CalcTransferTime.st ---- *)
(* ===========================================================================================
 *  STC_CalcTransferTime — Total transfer time calculation
 *
 *  Company : Galvatek part of the John Cockerill Group
 *  Author  : Jarmo Piipponen
 *  Created : 25.03.2026
 *
 * -------------------------------------------------------------------------------------------
 *  Calculates total transfer time between two stations using
 *  precomputed move time table plus operational delays:
 *  p2 = lift_s  + fromDroppingTime + dripTrayDelay
 *  p3 = travel_s
 *  p4 = sink_s  + dripTrayDelay    + toDeviceDelay
 *
 *  Lift station device_delay is NOT added because covers
 *  are opened during treatment time (overlaps).
 *
 *  All delay inputs are INT ×10 (tenths of second).
 *
 *  ------------------------------------------------------------------------------------------
 *
 *  Changes:
 *
 *
 *
 *)

FUNCTION STC_CalcTransferTime : REAL

(* Introduction of Variables ----------------------------------------------------------------*)

VAR_INPUT
  i_from_stn                : INT;     (* source station, e.g. 105 *)
  i_to_stn                  : INT;     (* destination station, e.g. 112 *)
  i_move                    : UDT_JC_MoveTimesType;   (* transporter's precomputed move times *)
  i_from_dropping_x10       : INT;     (* Stations[from].DrippingTime — tenths of second *)
  i_to_device_delay_x10     : INT;     (* Stations[to].DeviceDelay   — tenths of second *)
  i_drip_tray_delay_x10     : INT;     (* Transporters[trans].DripTrayDelay  — tenths of second *)
END_VAR

VAR
  from_idx                  : INT;
  to_idx                    : INT;
END_VAR

STC_CalcTransferTime := 0.0;
IF i_from_stn > 0 AND i_from_stn <> i_to_stn THEN
  from_idx := i_from_stn - MIN_STATION_INDEX;
  to_idx   := i_to_stn - MIN_STATION_INDEX;
  IF from_idx >= 1 AND from_idx <= 25 AND to_idx >= 1 AND to_idx <= 25 THEN
    STC_CalcTransferTime :=
      (* Phase 2: lift + dropping + drip tray *)
      INT_TO_REAL(i_move.LiftTime[from_idx]) / 10.0
      + INT_TO_REAL(i_from_dropping_x10) / 10.0
      + INT_TO_REAL(i_drip_tray_delay_x10) / 10.0
      (* Phase 3: horizontal travel *)
      + INT_TO_REAL(i_move.Travel[from_idx].ToTime[to_idx]) / 10.0
      (* Phase 4: sink + drip tray + device delay *)
      + INT_TO_REAL(i_move.SinkTime[to_idx]) / 10.0
      + INT_TO_REAL(i_drip_tray_delay_x10) / 10.0
      + INT_TO_REAL(i_to_device_delay_x10) / 10.0;
  END_IF;
END_IF;

END_FUNCTION

(* ---- STC_CollectActiveBatches.st ---- *)
(* ===========================================================================================
 *  STC_CollectActiveBatches — Filter active/waiting batches
 *
 *  Company : Galvatek part of the John Cockerill Group
 *  Author  : Jarmo Piipponen
 *  Created : 25.03.2026
 *
 * -------------------------------------------------------------------------------------------
 *  Returns count of matching batches; fills o_list via VAR_OUTPUT.
 *
 *  Mode:
 *  i_mode = 0 — active (in-production) batches
 *  i_mode = 1 — waiting batches (station 114 lookup)
 *
 *  ------------------------------------------------------------------------------------------
 *
 *  Changes:
 *
 *
 *
 *)

FUNCTION STC_CollectActiveBatches : INT   (* returns count *)

(* Introduction of Variables ----------------------------------------------------------------*)

VAR_INPUT
  i_mode                    : INT;    (* 0 = all active, 1 = waiting only *)
END_VAR

VAR_EXTERNAL CONSTANT
    MAX_UNITS               : INT;
    MAX_STATION_INDEX        : INT;
    USED                    : INT;
    TO_NONE                 : INT;
    NOT_PROCESSED           : INT;
    IN_PROCESS              : INT;
END_VAR

VAR_EXTERNAL
  g_batch                   : ARRAY[1..MAX_UNITS] OF UDT_BatchType;
  g_unit                    : ARRAY[1..MAX_UNITS] OF UDT_JC_UnitType;
  TreatmentPrograms                 : ARRAY[1..MAX_UNITS] OF UDT_TreatmentProgramType;
  g_station_occupancy             : ARRAY[1..MAX_STATION_INDEX] OF UDT_JC_UnitAtStationType;
END_VAR

VAR_OUTPUT
  o_list                    : ARRAY[1..MAX_UNITS] OF INT;  (* unit indices *)
END_VAR

VAR
  ui                        : INT;
  cnt                       : INT;
END_VAR

cnt := 0;
FOR ui := 1 TO MAX_UNITS DO
  o_list[ui] := 0;
END_FOR;

IF i_mode = 1 THEN
  (* ── Waiting batch: direct lookup at station 114 ── *)
  ui := g_station_occupancy[114].UnitId;
  IF ui >= 1 AND ui <= MAX_UNITS THEN
    IF g_unit[ui].Status = USED
       AND g_unit[ui].Target = TO_NONE
       AND g_batch[ui].State = NOT_PROCESSED
       AND g_batch[ui].ProgId = TreatmentPrograms[ui].ProgramId
       AND TreatmentPrograms[ui].ProgramId > 0 THEN
      cnt := 1;
      o_list[1] := ui;
    END_IF;
  END_IF;
  STC_CollectActiveBatches := cnt;
  RETURN;
END_IF;

(* ── Mode 0: active batches — loop ── *)
FOR ui := 1 TO MAX_UNITS DO
  IF g_unit[ui].Status = USED
     AND g_unit[ui].Target = TO_NONE
     AND g_batch[ui].ProgId = TreatmentPrograms[ui].ProgramId
     AND TreatmentPrograms[ui].ProgramId > 0 THEN

    IF g_batch[ui].State = IN_PROCESS
       AND g_batch[ui].CurStage >= 0
       AND g_batch[ui].CurStage <= 99 THEN
      cnt := cnt + 1;
      o_list[cnt] := ui;
    END_IF;
  END_IF;
END_FOR;

STC_CollectActiveBatches := cnt;

END_FUNCTION

(* ---- STC_CreateTasks.st ---- *)
(* ===========================================================================================
 *  STC_CreateTasks — Build task list from schedule for one unit
 *
 *  Company : Galvatek part of the John Cockerill Group
 *  Author  : Jarmo Piipponen
 *  Created : 25.03.2026
 *
 * -------------------------------------------------------------------------------------------
 *  Shared FC: both TSK and DEP call this with different arrays.
 *  Creates transporter tasks from the calculated schedule stages
 *  and appends them to the task queues.
 *
 *  ------------------------------------------------------------------------------------------
 *
 *  Changes:
 *
 *
 *
 *)

FUNCTION STC_CreateTasks : BOOL

(* Introduction of Variables ----------------------------------------------------------------*)

VAR_INPUT
  i_unit                    : INT;
END_VAR

VAR_IN_OUT  (* array sizes must match GVL_JC_Constants: 10=MAX_UNITS, 3=MAX_TRANSPORTERS *)
  io_schedule               : ARRAY[1..10] OF UDT_JC_TskScheduleType;
  io_task                   : ARRAY[1..3] OF UDT_JC_TskQueueType;
END_VAR

VAR_EXTERNAL CONSTANT
    MAX_TRANSPORTERS        : INT;
    MAX_UNITS               : INT;
    MAX_TASK_QUEUE          : INT;
    MIN_STATION_INDEX        : INT;
    MAX_STATION_INDEX        : INT;
END_VAR

VAR_EXTERNAL
  Transporters                     : ARRAY[0..MAX_TRANSPORTERS] OF UDT_TransporterType;
  Stations                 : ARRAY[MIN_STATION_INDEX..MAX_STATION_INDEX] OF UDT_StationType;
END_VAR

VAR
  si                        : INT;
  sc                        : INT;
  lift_stn                  : INT;
  sink_stn                  : INT;
  tid                       : INT;
  qi                        : INT;
  fb_find                   : STC_FindTransporter;
  eff_lift_stn              : INT;
END_VAR

STC_CreateTasks := FALSE;
IF i_unit < 1 OR i_unit > MAX_UNITS THEN RETURN; END_IF;

sc := io_schedule[i_unit].StageCount;
IF sc < 1 THEN RETURN; END_IF;

(* Start from 0 if Stages[0] exists (prepend), else from 1 *)
FOR si := 0 TO sc - 1 DO
  IF io_schedule[i_unit].Stages[si].station = 0 THEN
    (* Skip unused stage slot *)
  ELSE
    lift_stn := io_schedule[i_unit].Stages[si].station;
    sink_stn := io_schedule[i_unit].Stages[si + 1].station;

    IF lift_stn > 0 AND sink_stn > 0 THEN
      eff_lift_stn := lift_stn;
      IF lift_stn >= MIN_STATION_INDEX AND lift_stn <= MAX_STATION_INDEX
         AND sink_stn >= MIN_STATION_INDEX AND sink_stn <= MAX_STATION_INDEX THEN
        IF Stations[lift_stn].Crosstransport > 0
           AND Stations[lift_stn].ChangeStation > 0
           AND Stations[lift_stn].YPosition <> Stations[sink_stn].YPosition THEN
          eff_lift_stn := Stations[lift_stn].ChangeStation;
        END_IF;
      END_IF;

      fb_find(i_lift_stn := eff_lift_stn, i_sink_stn := sink_stn);
      tid := fb_find.o_trans;

      IF tid >= 1 AND tid <= 3 THEN
        qi := io_task[tid].Count + 1;
        IF qi <= MAX_TASK_QUEUE THEN
          io_task[tid].Queue[qi].Unit         := i_unit;
          io_task[tid].Queue[qi].Stage        := io_schedule[i_unit].Stages[si + 1].ProgramStage;
          io_task[tid].Queue[qi].SrcStage     := io_schedule[i_unit].Stages[si].ProgramStage;
          io_task[tid].Queue[qi].LiftStationTarget := eff_lift_stn;
          io_task[tid].Queue[qi].SinkStationTarget := sink_stn;
          io_task[tid].Queue[qi].StartTime   := io_schedule[i_unit].Stages[si].ExitTime;
          io_task[tid].Queue[qi].FinishTime  := io_schedule[i_unit].Stages[si + 1].EntryTime;
          io_task[tid].Queue[qi].CalcTime    := io_schedule[i_unit].Stages[si].CalcTime;
          io_task[tid].Queue[qi].MinTime     := io_schedule[i_unit].Stages[si].MinTime;
          io_task[tid].Queue[qi].MaxTime     := io_schedule[i_unit].Stages[si].MaxTime;
          io_task[tid].Count := qi;
        END_IF;
      END_IF;
    END_IF;
  END_IF; (* skip unused stage slot *)
END_FOR;

STC_CreateTasks := TRUE;

END_FUNCTION

(* ---- STC_DispatchTask.st ---- *)
(* ===========================================================================================
 *  STC_DispatchTask — Validate and dispatch tasks to transporters
 *
 *  Company : Galvatek part of the John Cockerill Group
 *  Author  : Jarmo Piipponen
 *  Created : 25.03.2026
 *
 * -------------------------------------------------------------------------------------------
 *  Called every PLC scan from MainScheduler.
 *  For each idle transporter with queued tasks:
 *  1. Skip if transporter not idle or queue empty
 *  2. Time check: start_time close enough?
 *  3. Sink station free check (with parallel alternatives)
 *  4. Conflict check against active transporters
 *  5. Dispatch: write to g_transporter → RunTasks picks it up
 *
 *  ------------------------------------------------------------------------------------------
 *
 *  Changes:
 *
 *
 *
 *)

FUNCTION STC_DispatchTask : BOOL

(* Introduction of Variables ----------------------------------------------------------------*)

VAR_EXTERNAL CONSTANT
    MAX_TRANSPORTERS        : INT;
    MAX_UNITS               : INT;
    MAX_STATIONS_PER_STEP   : INT;
    MAX_STEPS_PER_PROGRAM   : INT;
    MIN_STATION_INDEX        : INT;
    MAX_STATION_INDEX        : INT;
    SCH_DISPATCH_MARGIN_S   : REAL;
    USED                    : INT;
    PROCESSED               : INT;
END_VAR

VAR_EXTERNAL
  g_transporter             : ARRAY[1..MAX_TRANSPORTERS] OF UDT_TransporterStatusType;
  g_task                    : ARRAY[1..MAX_TRANSPORTERS] OF UDT_JC_TskQueueType;
  Stations                 : ARRAY[MIN_STATION_INDEX..MAX_STATION_INDEX] OF UDT_StationType;
  g_station_occupancy             : ARRAY[1..MAX_STATION_INDEX] OF UDT_JC_UnitAtStationType;
  g_unit                    : ARRAY[1..MAX_UNITS] OF UDT_JC_UnitType;
  TreatmentPrograms                 : ARRAY[1..MAX_UNITS] OF UDT_TreatmentProgramType;
  g_ntt                     : ARRAY[1..MAX_TRANSPORTERS] OF UDT_JC_NttTransporterType;
  g_batch                   : ARRAY[1..MAX_UNITS] OF UDT_BatchType;
  g_move                    : ARRAY[1..MAX_TRANSPORTERS] OF UDT_JC_MoveTimesType;
  Transporters                     : ARRAY[0..MAX_TRANSPORTERS] OF UDT_TransporterType;
  g_schedule                : ARRAY[1..MAX_UNITS] OF UDT_JC_TskScheduleType;
  g_time_s                  : LINT;
  g_event_pending           : UDT_JC_EventMsgType;
  g_event_pending_valid     : BOOL;
  g_dispatched_task         : ARRAY[1..MAX_TRANSPORTERS] OF UDT_JC_DispatchedTaskType;
END_VAR

VAR
  ti                        : INT;     (* transporter loop *)
  (* Task fields — read from queue[1] to avoid struct copy *)
  t_unit                    : INT;
  t_stage                   : INT;
  t_lift                    : INT;
  t_sink                    : INT;
  t_start                   : LINT;
  t_finish                  : LINT;
  t_calc_time               : DINT;
  (* Time check *)
  travel_s                  : REAL;
  margin_s                  : LINT;
  from_idx                  : INT;
  to_idx                    : INT;
  (* Sink search *)
  sink_stn                  : INT;
  sink_free                 : BOOL;
  best_stn                  : INT;
  best_change               : LINT;
  si                        : INT;
  cand_stn                  : INT;
  cand_free                 : BOOL;
  uj                        : INT;
  tgt                       : INT;
  ntt_idx                   : INT;     (* resolved NTT index (buffer 6/7/8) *)
  ntt_cnt                   : INT;
  ntt_fb_cnt                : INT;
  (* Conflict check *)
  conflict                  : BOOL;
  cj                        : INT;
  task_min                  : INT;     (* min station of our proposed task *)
  task_max                  : INT;     (* max station of our proposed task *)
  (* Queue position loop *)
  qi                        : INT;
  (* Shift-down after dispatch *)
  sh                        : INT;
  (* Transfer time for batch progress bar *)
  xfer_total                : REAL;
  (* Program stage number for event *)
  prog_stage                : INT;
  (* Manual task dispatch flag *)
  unit_ok                   : BOOL;
END_VAR

FOR ti := 1 TO MAX_TRANSPORTERS DO

  (* ── 1. Skip if not idle or queue empty ── *)
  (* Accept idle (Phase=0) OR move-away in progress (Phase=1, Status=3) *)
  IF (g_transporter[ti].Phase = 0 OR (g_transporter[ti].Phase = 1 AND g_transporter[ti].Status = 3))
     AND g_task[ti].Count >= 1 THEN

    (* Try each queue position — skip blocked tasks, dispatch first feasible *)
    FOR qi := 1 TO g_task[ti].Count DO

    (* Read task fields from queue position qi *)
    t_unit      := g_task[ti].Queue[qi].Unit;
    t_stage     := g_task[ti].Queue[qi].Stage;  (* schedule index *)
    t_lift      := g_task[ti].Queue[qi].LiftStationTarget;
    t_sink      := g_task[ti].Queue[qi].SinkStationTarget;
    t_start     := g_task[ti].Queue[qi].StartTime;
    t_finish    := g_task[ti].Queue[qi].FinishTime;
    t_calc_time := g_task[ti].Queue[qi].CalcTime;

    (* Queue[].Stage already contains ProgramStage (set by STC_CreateTasks) *)
    prog_stage := t_stage;

    (* ── 1b. Lift station unit check — unit must be AT the lift station ── *)
    (* Manual tasks have Unit=0 → skip unit-location check *)
    (* NOTE: CODESYS does NOT short-circuit OR — use nested IFs *)
    unit_ok := FALSE;
    IF t_unit = 0 THEN
      unit_ok := TRUE;
    ELSIF t_unit >= 1 AND t_unit <= MAX_UNITS THEN
      IF g_unit[t_unit].location = t_lift THEN
        unit_ok := TRUE;
      END_IF;
    END_IF;

    IF unit_ok THEN

    (* ── 2. Time check ── *)
    travel_s := 0.0;
    IF g_transporter[ti].CurrentStation > 0 AND t_lift > 0
       AND g_transporter[ti].CurrentStation <> t_lift THEN
      from_idx := g_transporter[ti].CurrentStation - MIN_STATION_INDEX;
      to_idx   := t_lift - MIN_STATION_INDEX;
      IF from_idx >= 1 AND from_idx <= 30 AND to_idx >= 1 AND to_idx <= 30 THEN
        travel_s := INT_TO_REAL(g_move[ti].Travel[from_idx].ToTime[to_idx]) / 10.0;
      END_IF;
    END_IF;

    margin_s := t_start - g_time_s;

    IF margin_s <= REAL_TO_LINT(travel_s + SCH_DISPATCH_MARGIN_S) THEN

      (* ── 3. Sink station free check ── *)
      sink_stn := t_sink;
      sink_free := FALSE;

      IF sink_stn >= MIN_STATION_INDEX AND sink_stn <= MAX_STATION_INDEX THEN
        sink_free := TRUE;
        FOR uj := 1 TO MAX_UNITS DO
          IF g_unit[uj].location = sink_stn AND g_unit[uj].Status = USED THEN
            sink_free := FALSE;
          END_IF;
        END_FOR;
      END_IF;

      IF NOT sink_free THEN
        (* Search alternative parallel stations *)
        best_stn := 0;
        best_change := LINT#2000000000;

        IF prog_stage >= 1 AND prog_stage <= MAX_STEPS_PER_PROGRAM
           AND t_unit >= 1 AND t_unit <= MAX_UNITS THEN
          (* Treatment task — look in TreatmentPrograms for parallel stations *)
          FOR si := 0 TO MAX_STATIONS_PER_STEP - 1 DO
            cand_stn := TreatmentPrograms[t_unit].Steps[prog_stage].Stations[si];
            IF cand_stn > 0 AND cand_stn <> t_sink THEN
              IF cand_stn >= MIN_STATION_INDEX AND cand_stn <= MAX_STATION_INDEX THEN
                cand_free := TRUE;
                FOR uj := 1 TO MAX_UNITS DO
                  IF g_unit[uj].location = cand_stn AND g_unit[uj].Status = USED THEN
                    cand_free := FALSE;
                  END_IF;
                END_FOR;
                IF cand_free THEN
                  IF g_station_occupancy[cand_stn].ChangeTime < best_change THEN
                    best_change := g_station_occupancy[cand_stn].ChangeTime;
                    best_stn := cand_stn;
                  END_IF;
                END_IF;
              END_IF;
            END_IF;
          END_FOR;

        ELSIF prog_stage = 0 AND t_unit >= 1 AND t_unit <= MAX_UNITS THEN
          (* No-treatment task — look in g_ntt for alternatives *)
          tgt := g_unit[t_unit].Target;
          IF tgt >= 1 AND tgt <= 5 THEN
            (* Resolve buffer NTT index like NoTreatment does *)
            IF tgt = 2 THEN
              IF g_batch[t_unit].BatchCode = 0 THEN
                ntt_idx := 6;
              ELSIF g_batch[t_unit].State = PROCESSED THEN
                ntt_idx := 8;
              ELSE
                ntt_idx := 7;
              END_IF;
            ELSE
              ntt_idx := tgt;
            END_IF;
            (* Check primary stations *)
            ntt_cnt := g_ntt[ti].Target[ntt_idx].StationCount;
            FOR si := 1 TO ntt_cnt DO
              IF si <= MAX_STATIONS_PER_STEP THEN
                cand_stn := g_ntt[ti].Target[ntt_idx].Stations[si];
                IF cand_stn > 0 AND cand_stn <> t_sink THEN
                  IF cand_stn >= MIN_STATION_INDEX AND cand_stn <= MAX_STATION_INDEX THEN
                    cand_free := TRUE;
                    FOR uj := 1 TO MAX_UNITS DO
                      IF g_unit[uj].location = cand_stn AND g_unit[uj].Status = USED THEN
                        cand_free := FALSE;
                      END_IF;
                    END_FOR;
                    IF cand_free THEN
                      IF g_station_occupancy[cand_stn].ChangeTime < best_change THEN
                        best_change := g_station_occupancy[cand_stn].ChangeTime;
                        best_stn := cand_stn;
                      END_IF;
                    END_IF;
                  END_IF;
                END_IF;
              END_IF;
            END_FOR;
            (* Check fallback stations *)
            ntt_fb_cnt := g_ntt[ti].Target[ntt_idx].FallbackCount;
            FOR si := 1 TO ntt_fb_cnt DO
              IF si <= MAX_STATIONS_PER_STEP THEN
                cand_stn := g_ntt[ti].Target[ntt_idx].FallbackStations[si];
                IF cand_stn > 0 AND cand_stn <> t_sink THEN
                  IF cand_stn >= MIN_STATION_INDEX AND cand_stn <= MAX_STATION_INDEX THEN
                    cand_free := TRUE;
                    FOR uj := 1 TO MAX_UNITS DO
                      IF g_unit[uj].location = cand_stn AND g_unit[uj].Status = USED THEN
                        cand_free := FALSE;
                      END_IF;
                    END_FOR;
                    IF cand_free THEN
                      IF g_station_occupancy[cand_stn].ChangeTime < best_change THEN
                        best_change := g_station_occupancy[cand_stn].ChangeTime;
                        best_stn := cand_stn;
                      END_IF;
                    END_IF;
                  END_IF;
                END_IF;
              END_IF;
            END_FOR;
          END_IF;
        END_IF;

        IF best_stn > 0 THEN
          sink_stn := best_stn;
          sink_free := TRUE;
        END_IF;
      END_IF;  (* NOT sink_free *)

      IF sink_free THEN

        (* ── 4. Conflict check ── *)
        conflict := FALSE;

        IF t_lift <= sink_stn THEN
          task_min := t_lift;
          task_max := sink_stn;
        ELSE
          task_min := sink_stn;
          task_max := t_lift;
        END_IF;

        FOR cj := 1 TO MAX_TRANSPORTERS DO
          IF cj <> ti AND g_transporter[cj].Phase > 0 THEN

            (* a) T2's entire active task inside our range → conflict *)
            IF g_transporter[cj].LiftStationTarget >= task_min
               AND g_transporter[cj].LiftStationTarget <= task_max
               AND g_transporter[cj].SinkStationTarget >= task_min
               AND g_transporter[cj].SinkStationTarget <= task_max THEN
              conflict := TRUE;
            END_IF;

            (* b) T2 delivers to one of our exact stations → conflict *)
            IF g_transporter[cj].SinkStationTarget = t_lift
               OR g_transporter[cj].SinkStationTarget = sink_stn THEN
              conflict := TRUE;
            END_IF;

          END_IF;
        END_FOR;

        IF NOT conflict THEN
          (* ── 5. Dispatch: assign task to transporter ── *)
          g_transporter[ti].TaskId      := t_start;
          g_transporter[ti].LiftStationTarget := t_lift;
          g_transporter[ti].SinkStationTarget := sink_stn;
          g_transporter[ti].CurrentTaskFinishTime := g_task[ti].Queue[qi].FinishTime;
          g_station_occupancy[ti].UnitId      := t_unit;
          g_transporter[ti].TaskRemainingTime := t_calc_time;

          (* ── 5b. Fill dispatched task package ── *)
          g_dispatched_task[ti].TaskId           := t_start;
          g_dispatched_task[ti].UnitId           := t_unit;
          g_dispatched_task[ti].LiftStation      := t_lift;
          g_dispatched_task[ti].SinkStation      := sink_stn;
          IF t_lift >= MIN_STATION_INDEX AND t_lift <= MAX_STATION_INDEX THEN
            g_dispatched_task[ti].LiftX              := Stations[t_lift].XPosition;
            g_dispatched_task[ti].LiftKind           := Stations[t_lift].DryWet;
            g_dispatched_task[ti].DroppingTime_x10   := Stations[t_lift].DrippingTime;
            g_dispatched_task[ti].LiftDeviceDelay_x10 := Stations[t_lift].DeviceDelay;
          END_IF;
          IF sink_stn >= MIN_STATION_INDEX AND sink_stn <= MAX_STATION_INDEX THEN
            g_dispatched_task[ti].SinkX              := Stations[sink_stn].XPosition;
            g_dispatched_task[ti].SinkKind           := Stations[sink_stn].DryWet;
            g_dispatched_task[ti].SinkDeviceDelay_x10 := Stations[sink_stn].DeviceDelay;
          END_IF;
          g_dispatched_task[ti].DripTrayDelay_x10 := Transporters[ti].DripTrayDelay;
          g_dispatched_task[ti].TreatmentTime    := t_calc_time;
          g_dispatched_task[ti].MinTime          := g_task[ti].Queue[qi].MinTime;
          g_dispatched_task[ti].MaxTime          := g_task[ti].Queue[qi].MaxTime;
          g_dispatched_task[ti].NttPrimary       := g_task[ti].Queue[qi].NttPrimary;
          IF t_unit >= 1 AND t_unit <= MAX_UNITS THEN
            g_dispatched_task[ti].BatchCode      := g_batch[t_unit].BatchCode;
            g_dispatched_task[ti].ProgramStage   := g_batch[t_unit].CurStage;
          ELSE
            g_dispatched_task[ti].BatchCode      := 0;
            g_dispatched_task[ti].ProgramStage   := 0;
          END_IF;
          g_dispatched_task[ti].Active           := TRUE;

          (* ── Emit TASK_DISPATCHED event (msg_type=1) ── *)
          xfer_total := STC_CalcTransferTime(
            i_from_stn            := t_lift,
            i_to_stn              := sink_stn,
            i_move                := g_move[ti],
            i_from_dropping_x10   := Stations[t_lift].DrippingTime,
            i_to_device_delay_x10 := Stations[sink_stn].DeviceDelay,
            i_drip_tray_delay_x10 := Transporters[ti].DripTrayDelay
          );
          IF xfer_total < 1.0 THEN
            xfer_total := INT_TO_REAL(ABS(sink_stn - t_lift)) * 8.0;
          END_IF;
  IF xfer_total < 5.0 THEN xfer_total := 60.0; END_IF;
          g_dispatched_task[ti].TransferTime_x10 := REAL_TO_DINT(xfer_total * 10.0);
          IF NOT g_event_pending_valid THEN
            g_event_pending.MsgType := 1;
            g_event_pending.TsHi := LINT_TO_UINT(g_time_s / LINT#65536);
            g_event_pending.TsLo := LINT_TO_UINT(g_time_s MOD LINT#65536);
            g_event_pending.Payload[1]  := LINT_TO_INT(t_start / LINT#65536);   (* TaskId_Hi *)
            g_event_pending.Payload[2]  := LINT_TO_INT(t_start MOD LINT#65536);  (* TaskId_Lo *)
            g_event_pending.Payload[3]  := ti;
            g_event_pending.Payload[4]  := t_unit;
            g_event_pending.Payload[5]  := t_lift;
            g_event_pending.Payload[6]  := sink_stn;
            IF t_unit >= 1 AND t_unit <= MAX_UNITS THEN
              prog_stage := g_batch[t_unit].CurStage;
              g_event_pending.Payload[7]  := prog_stage;
              g_event_pending.Payload[8]  := g_batch[t_unit].BatchCode;
            ELSE
              g_event_pending.Payload[7]  := 0;
              g_event_pending.Payload[8]  := 0;
            END_IF;
            g_event_pending.Payload[9]  := DINT_TO_INT(t_calc_time);
            g_event_pending.Payload[10] := DINT_TO_INT(g_task[ti].Queue[qi].MinTime);
            g_event_pending.Payload[11] := DINT_TO_INT(g_task[ti].Queue[qi].MaxTime);
            g_event_pending.Payload[12] := REAL_TO_INT(xfer_total);
            g_event_pending_valid := TRUE;
          END_IF;

          (* Copy station-specific timing from config *)
          IF t_lift >= MIN_STATION_INDEX AND t_lift <= MAX_STATION_INDEX THEN
            g_transporter[ti].DrippingTime := Stations[t_lift].DrippingTime;
          END_IF;

          (* Shift queue: remove position qi, move rest up *)
          FOR sh := qi + 1 TO g_task[ti].Count DO
            g_task[ti].Queue[sh - 1] := g_task[ti].Queue[sh];
          END_FOR;
          (* Clear last slot *)
          g_task[ti].Queue[g_task[ti].Count].Unit := 0;
          g_task[ti].Queue[g_task[ti].Count].Stage := 0;
          g_task[ti].Queue[g_task[ti].Count].SrcStage := 0;
          g_task[ti].Queue[g_task[ti].Count].LiftStationTarget := 0;
          g_task[ti].Queue[g_task[ti].Count].SinkStationTarget := 0;
          g_task[ti].Queue[g_task[ti].Count].StartTime := 0;
          g_task[ti].Queue[g_task[ti].Count].FinishTime := 0;
          g_task[ti].Queue[g_task[ti].Count].CalcTime := 0;
          g_task[ti].Queue[g_task[ti].Count].MinTime := 0;
          g_task[ti].Queue[g_task[ti].Count].MaxTime := 0;
          g_task[ti].Count := g_task[ti].Count - 1;
          EXIT;  (* dispatched — stop searching this queue *)

        END_IF;  (* NOT conflict *)

      END_IF;  (* sink_free *)

    END_IF;  (* time check *)

    END_IF;  (* unit at lift station *)

    END_FOR;  (* qi — try next queue position *)

  END_IF;  (* idle + queue *)

END_FOR;

STC_DispatchTask := TRUE;

END_FUNCTION

(* ---- STC_FC_CalcHorizontalTravel.st ---- *)
(* ===========================================================================================
 *  STC_FC_CalcHorizontalTravel — Horizontal travel time
 *
 *  Company : Galvatek part of the John Cockerill Group
 *  Author  : Jarmo Piipponen
 *  Created : 25.03.2026
 *
 * -------------------------------------------------------------------------------------------
 *  Calculates horizontal travel time between two stations
 *  (no lift/sink) using precomputed move time table.
 *  Caller passes iMove (UDT_JC_MoveTimesType) for the
 *  specific transporter.
 *
 *  ------------------------------------------------------------------------------------------
 *
 *  Changes:
 *
 *
 *
 *)

FUNCTION STC_FC_CalcHorizontalTravel : REAL

(* Introduction of Variables ----------------------------------------------------------------*)

VAR_INPUT
  iFromStn                : INT;     (* source station number *)
  iToStn                  : INT;     (* destination station number *)
  iMove                    : UDT_JC_MoveTimesType;   (* transporter's precomputed move times *)
END_VAR

VAR
  vFromIdx                  : INT;
  vToIdx                    : INT;
END_VAR

STC_FC_CalcHorizontalTravel := 0.0;
IF iFromStn > 0 AND iToStn > 0 AND iFromStn <> iToStn THEN
  vFromIdx := iFromStn - MIN_STATION_INDEX;
  vToIdx   := iToStn - MIN_STATION_INDEX;
  IF vFromIdx >= 1 AND vFromIdx <= 25 AND vToIdx >= 1 AND vToIdx <= 25 THEN
    STC_FC_CalcHorizontalTravel := INT_TO_REAL(iMove.Travel[vFromIdx].ToTime[vToIdx]) / 10.0;
  END_IF;
END_IF;

END_FUNCTION

(* ---- STC_FC_CalcSchedule.st ---- *)
(* ===========================================================================================
 *  STC_FC_CalcSchedule — Calculate batch schedule for one unit
 *
 *  Company : Galvatek part of the John Cockerill Group
 *  Author  : Jarmo Piipponen
 *  Created : 25.03.2026
 *
 * -------------------------------------------------------------------------------------------
 *  Shared FC: both TSK and DEP call this with different arrays.
 *  Calculates start/finish times for each treatment stage based
 *  on elapsed time, cal_time and transfer durations.
 *
 *  ------------------------------------------------------------------------------------------
 *
 *  Changes:
 *
 *
 *
 *)

FUNCTION STC_FC_CalcSchedule : BOOL

(* Introduction of Variables ----------------------------------------------------------------*)

VAR_INPUT
  iUnit                    : INT;
  iTrans                   : INT;
  iTimeS                  : LINT;
END_VAR

VAR_IN_OUT  (* array sizes must match GVL_JC_Constants: 10=MAX_UNITS *)
  ioSchedule               : ARRAY[1..10] OF UDT_JC_TskScheduleType;
  ioBatch                  : ARRAY[1..10] OF UDT_BatchType;
  ioProgram                : ARRAY[1..10] OF UDT_TreatmentProgramType;
END_VAR

VAR_EXTERNAL CONSTANT
    MIN_STATION_INDEX        : INT;
    MAX_STATION_INDEX        : INT;
    MAX_UNITS               : INT;
    MAX_TRANSPORTERS        : INT;
    MAX_STEPS_PER_PROGRAM   : INT;
    NOT_PROCESSED           : INT;
    USED                    : INT;
END_VAR

VAR_EXTERNAL
  Unit                    : ARRAY[1..MAX_UNITS] OF UDT_JC_UnitType;
  Stations                 : ARRAY[MIN_STATION_INDEX..MAX_STATION_INDEX] OF UDT_StationType;
  StationOccupancy             : ARRAY[1..MAX_STATION_INDEX] OF UDT_JC_UnitAtStationType;
  CountStations              : INT;
  Move                    : ARRAY[1..MAX_TRANSPORTERS] OF UDT_JC_MoveTimesType;
  Transporters                     : ARRAY[0..MAX_TRANSPORTERS] OF UDT_TransporterType;
  TransporterStatus             : ARRAY[1..MAX_TRANSPORTERS] OF UDT_TransporterStatusType;
END_VAR

VAR
  vStg                       : INT;
  vStnNum                   : INT;
  vPrevStn                  : INT;
  vCurStage                 : INT;
  vLocation                  : INT;
  vStartSt                  : INT;
  vEntryT                   : LINT;
  vExitT                    : LINT;
  vXferT                    : REAL;
  vCalcS                    : REAL;
  vMinS                     : REAL;
  vMaxS                     : REAL;
  vIsOnStn                 : BOOL;
  vIsFirst                  : BOOL;
  vRemainS                  : REAL;
  vElapsedS                 : REAL;
  vP                         : INT;
  vChosenStn                : INT;
  vTmpMove                  : UDT_JC_MoveTimesType;
  vCandArr                  : ARRAY[1..5] OF INT;
  vCandCnt                  : INT;
  vSchedOccupied            : ARRAY[1..5] OF BOOL;
  vBestChangeTime          : LINT;
  vMyEntry                  : LINT;
  vMyExit                   : LINT;
  vOvStart                  : LINT;
  vOvEnd                    : LINT;
  vUj                        : INT;
  vSj                        : INT;
END_VAR

STC_FC_CalcSchedule := FALSE;
IF iUnit < 1 OR iUnit > MAX_UNITS THEN RETURN; END_IF;
IF iTrans < 1 OR iTrans > MAX_TRANSPORTERS THEN RETURN; END_IF;

vCurStage := ioBatch[iUnit].CurStage;
vLocation  := Unit[iUnit].vLocation;
vIsOnStn := vLocation >= MIN_STATION_INDEX;

(* Clear old schedule *)
FOR vStg := 0 TO MAX_STEPS_PER_PROGRAM DO
  ioSchedule[iUnit].Stages[vStg].station := 0;
  ioSchedule[iUnit].Stages[vStg].ProgramStage := 0;
  ioSchedule[iUnit].Stages[vStg].EntryTime := 0;
  ioSchedule[iUnit].Stages[vStg].ExitTime := 0;
  ioSchedule[iUnit].Stages[vStg].MinTime := 0;
  ioSchedule[iUnit].Stages[vStg].CalcTime := 0;
  ioSchedule[iUnit].Stages[vStg].MaxTime := 0;
  ioSchedule[iUnit].Stages[vStg].TransferTime := 0;
END_FOR;
ioSchedule[iUnit].StageCount := 0;

(* Waiting batch (state = NOT_PROCESSED): treat as stage 0 *)
IF ioBatch[iUnit].State = NOT_PROCESSED THEN
  vCurStage := 0;
END_IF;

IF vIsOnStn THEN
  vStartSt := vCurStage;
ELSE
  vStartSt := vCurStage + 1;
END_IF;
IF vStartSt < 1 THEN
  vStartSt := 1;
END_IF;

IF vIsOnStn THEN
  vPrevStn := vLocation;
ELSIF vCurStage >= 1 AND vCurStage <= 30 THEN
  vPrevStn := ioProgram[iUnit].Steps[vCurStage].Stations[0];
ELSE
  vPrevStn := 0;
END_IF;

vExitT := iTimeS;
vIsFirst := TRUE;

(* Prepend current vLocation to Stages[0] when unit needs pre-positioning *)
IF vIsOnStn AND vStartSt >= 1 THEN
  vStnNum := 0;
  FOR vP := 0 TO 4 DO
    IF ioProgram[iUnit].Steps[vStartSt].Stations[vP] = vLocation THEN
      vStnNum := vLocation;
    END_IF;
  END_FOR;
  IF vStnNum = 0 THEN
    ioSchedule[iUnit].Stages[0].station       := vLocation;
    ioSchedule[iUnit].Stages[0].ProgramStage := 0;
    ioSchedule[iUnit].Stages[0].EntryTime    := vExitT;
    ioSchedule[iUnit].Stages[0].TransferTime := 0;

    IF ioBatch[iUnit].CurStage = 0 AND ioBatch[iUnit].CalTime > 0 THEN
      IF ioBatch[iUnit].StartTime > 0 AND ioBatch[iUnit].StartTime < iTimeS THEN
        vElapsedS := LINT_TO_REAL(iTimeS - ioBatch[iUnit].StartTime);
      ELSE
        vElapsedS := 0.0;
      END_IF;
      vRemainS := DINT_TO_REAL(ioBatch[iUnit].CalTime) - vElapsedS;
  IF vRemainS < 1.0 THEN vRemainS := 1.0; END_IF;
      vExitT := iTimeS + REAL_TO_LINT(vRemainS);
      ioSchedule[iUnit].Stages[0].ExitTime  := vExitT;
      ioSchedule[iUnit].Stages[0].CalcTime  := REAL_TO_DINT(vRemainS);
      ioSchedule[iUnit].Stages[0].MinTime   := ioBatch[iUnit].MinTime;
      ioSchedule[iUnit].Stages[0].MaxTime   := ioBatch[iUnit].MaxTime;
    ELSE
      (* Pickup wait: transporter horizontal travel time to this station, min 5s *)
      vCalcS := STC_FC_CalcHorizontalTravel(
        iFromStn := TransporterStatus[iTrans].CurrentStation,
        iToStn   := vLocation,
        iMove     := Move[iTrans]);
      IF vCalcS < 5.0 THEN vCalcS := 5.0; END_IF;
      vExitT := iTimeS + REAL_TO_LINT(vCalcS);
      ioSchedule[iUnit].Stages[0].ExitTime  := vExitT;
      ioSchedule[iUnit].Stages[0].CalcTime  := REAL_TO_DINT(vCalcS);
      ioSchedule[iUnit].Stages[0].MinTime   := REAL_TO_DINT(vCalcS);
      ioSchedule[iUnit].Stages[0].MaxTime   := REAL_TO_DINT(2.0 * vCalcS);
    END_IF;

    vIsFirst := FALSE;
  END_IF;
END_IF;

(* ============================================================
   MAIN LOOP: Calculate schedule for each program stage
   ============================================================ *)
FOR vStg := vStartSt TO ioProgram[iUnit].StepCount DO

  vCandCnt := 0;
  FOR vP := 0 TO 4 DO
    IF ioProgram[iUnit].Steps[vStg].Stations[vP] > 0 THEN
      vCandCnt := vCandCnt + 1;
      vCandArr[vCandCnt] := ioProgram[iUnit].Steps[vStg].Stations[vP];
      vSchedOccupied[vCandCnt] := FALSE;
    END_IF;
  END_FOR;

  IF vCandCnt = 0 THEN
    EXIT;
  END_IF;

  vChosenStn := 0;
  IF vIsFirst AND vIsOnStn AND vStg = vCurStage THEN
    FOR vP := 1 TO vCandCnt DO
      IF vCandArr[vP] = vLocation THEN
        vChosenStn := vLocation;
      END_IF;
    END_FOR;
  END_IF;

  IF vChosenStn = 0 THEN
    IF vCandCnt = 1 THEN
      vChosenStn := vCandArr[1];
    ELSE
      (* Estimate this batch's time window per candidate for overlap check *)
      vCalcS := DINT_TO_REAL(ioProgram[iUnit].Steps[vStg].CalTime);
      vTmpMove := Move[iTrans];

      FOR vP := 1 TO vCandCnt DO
        (* Calculate entry/exit per candidate station individually *)
        vXferT := STC_FC_CalcTransferTime(
          iFromStn            := vPrevStn,
          iToStn              := vCandArr[vP],
          iMove                := vTmpMove,
          iFromDroppingX10   := Stations[vPrevStn].DrippingTime,
          iToDeviceDelayX10 := Stations[vCandArr[vP]].DeviceDelay,
          iDripTrayDelayX10 := Transporters[iTrans].DripTrayDelay
        );
        vMyEntry := vExitT + REAL_TO_LINT(vXferT);
        vMyExit  := vMyEntry + REAL_TO_LINT(vCalcS);

        FOR vUj := 1 TO MAX_UNITS DO
          IF vUj <> iUnit AND ioSchedule[vUj].StageCount > 0 THEN
            FOR vSj := 0 TO ioSchedule[vUj].StageCount DO
              IF ioSchedule[vUj].Stages[vSj].station = vCandArr[vP] THEN
                vOvStart := vMyEntry;
                IF ioSchedule[vUj].Stages[vSj].EntryTime > vOvStart THEN
                  vOvStart := ioSchedule[vUj].Stages[vSj].EntryTime;
                END_IF;
                vOvEnd := vMyExit;
                IF ioSchedule[vUj].Stages[vSj].ExitTime < vOvEnd THEN
                  vOvEnd := ioSchedule[vUj].Stages[vSj].ExitTime;
                END_IF;
                IF vOvEnd > vOvStart THEN
                  vSchedOccupied[vP] := TRUE;
                END_IF;
              END_IF;
            END_FOR;
          END_IF;
        END_FOR;

      END_FOR;

      (* Pass 1: prefer schedule-free station, pick earliest ChangeTime *)
      vBestChangeTime := LINT#9999999999;
      FOR vP := 1 TO vCandCnt DO
        IF NOT vSchedOccupied[vP] THEN
          IF vCandArr[vP] >= MIN_STATION_INDEX AND vCandArr[vP] <= MAX_STATION_INDEX THEN
            IF StationOccupancy[vCandArr[vP]].ChangeTime < vBestChangeTime THEN
              vBestChangeTime := StationOccupancy[vCandArr[vP]].ChangeTime;
              vChosenStn := vCandArr[vP];
            END_IF;
          END_IF;
        END_IF;
      END_FOR;

      (* Pass 2: all sched-occupied — pick first candidate *)
      IF vChosenStn = 0 THEN
        vChosenStn := vCandArr[1];
      END_IF;
    END_IF;
  END_IF;

  vStnNum := vChosenStn;

  vCalcS := DINT_TO_REAL(ioProgram[iUnit].Steps[vStg].CalTime);
  vMinS  := DINT_TO_REAL(ioProgram[iUnit].Steps[vStg].MinTime);
  vMaxS  := DINT_TO_REAL(ioProgram[iUnit].Steps[vStg].MaxTime);

  vTmpMove := Move[iTrans];
  IF vPrevStn >= MIN_STATION_INDEX AND vPrevStn <= MAX_STATION_INDEX
     AND vStnNum >= MIN_STATION_INDEX AND vStnNum <= MAX_STATION_INDEX THEN
    IF Stations[vPrevStn].Crosstransport > 0
       AND Stations[vPrevStn].ChangeStation > 0
       AND Stations[vPrevStn].YPosition <> Stations[vStnNum].YPosition THEN
      vXferT := INT_TO_REAL(Stations[vPrevStn].CrossTransportTime)
              + STC_FC_CalcTransferTime(
                  iFromStn            := Stations[vPrevStn].ChangeStation,
                  iToStn              := vStnNum,
                  iMove                := vTmpMove,
                  iFromDroppingX10   := Stations[Stations[vPrevStn].ChangeStation].DrippingTime,
                  iToDeviceDelayX10 := Stations[vStnNum].DeviceDelay,
                  iDripTrayDelayX10 := Transporters[iTrans].DripTrayDelay
                );
    ELSE
      vXferT := STC_FC_CalcTransferTime(
        iFromStn            := vPrevStn,
        iToStn              := vStnNum,
        iMove                := vTmpMove,
        iFromDroppingX10   := Stations[vPrevStn].DrippingTime,
        iToDeviceDelayX10 := Stations[vStnNum].DeviceDelay,
        iDripTrayDelayX10 := Transporters[iTrans].DripTrayDelay
      );
    END_IF;
  ELSE
    vXferT := 60.0;
  END_IF;

  IF vIsFirst AND vIsOnStn AND vStg = vCurStage THEN
    vEntryT := iTimeS;
    IF ioBatch[iUnit].StartTime > 0 THEN
      vElapsedS := LINT_TO_REAL(iTimeS - ioBatch[iUnit].StartTime);
    ELSE
      vElapsedS := 0.0;
    END_IF;
    vRemainS := DINT_TO_REAL(ioBatch[iUnit].CalTime) - vElapsedS;
  IF vRemainS < 1.0 THEN vRemainS := 1.0; END_IF;
    vExitT := iTimeS + REAL_TO_LINT(vRemainS);
  ELSIF vIsFirst AND NOT vIsOnStn THEN
    IF ioBatch[iUnit].StartTime > 0 AND ioBatch[iUnit].CalTime > 0 THEN
      vEntryT := ioBatch[iUnit].StartTime + DINT_TO_LINT(ioBatch[iUnit].CalTime);
    ELSE
      vEntryT := iTimeS + REAL_TO_LINT(vXferT);
    END_IF;
    vExitT  := vEntryT + REAL_TO_LINT(vCalcS);
  ELSE
    vEntryT := vExitT + REAL_TO_LINT(vXferT);
    vExitT  := vEntryT + REAL_TO_LINT(vCalcS);
  END_IF;

  IF vStg <= 30 THEN
    ioSchedule[iUnit].Stages[vStg].station       := vStnNum;
    ioSchedule[iUnit].Stages[vStg].ProgramStage := vStg;
    ioSchedule[iUnit].Stages[vStg].EntryTime    := vEntryT;
    ioSchedule[iUnit].Stages[vStg].ExitTime     := vExitT;
    ioSchedule[iUnit].Stages[vStg].MinTime      := REAL_TO_DINT(vMinS);
    ioSchedule[iUnit].Stages[vStg].CalcTime     := REAL_TO_DINT(vCalcS);
    ioSchedule[iUnit].Stages[vStg].MaxTime      := REAL_TO_DINT(vMaxS);
    ioSchedule[iUnit].Stages[vStg].TransferTime := REAL_TO_DINT(vXferT);
    ioSchedule[iUnit].StageCount := vStg;
  END_IF;

  vPrevStn := vStnNum;
  vIsFirst := FALSE;

END_FOR;

STC_FC_CalcSchedule := TRUE;

END_FUNCTION

(* ---- STC_FC_CalcTransferTime.st ---- *)
(* ===========================================================================================
 *  STC_FC_CalcTransferTime — Total transfer time calculation
 *
 *  Company : Galvatek part of the John Cockerill Group
 *  Author  : Jarmo Piipponen
 *  Created : 25.03.2026
 *
 * -------------------------------------------------------------------------------------------
 *  Calculates total transfer time between two stations using
 *  precomputed move time table plus operational delays:
 *  p2 = lift_s  + fromDroppingTime + dripTrayDelay
 *  p3 = travel_s
 *  p4 = sink_s  + dripTrayDelay    + toDeviceDelay
 *
 *  Lift station device_delay is NOT added because covers
 *  are opened during treatment time (overlaps).
 *
 *  All delay inputs are INT ×10 (tenths of second).
 *
 *  ------------------------------------------------------------------------------------------
 *
 *  Changes:
 *
 *
 *
 *)

FUNCTION STC_FC_CalcTransferTime : REAL

(* Introduction of Variables ----------------------------------------------------------------*)

VAR_INPUT
  iFromStn                : INT;     (* source station, e.g. 105 *)
  iToStn                  : INT;     (* destination station, e.g. 112 *)
  iMove                    : UDT_JC_MoveTimesType;   (* transporter's precomputed move times *)
  iFromDroppingX10       : INT;     (* Stations[from].DrippingTime — tenths of second *)
  iToDeviceDelayX10     : INT;     (* Stations[to].DeviceDelay   — tenths of second *)
  iDripTrayDelayX10     : INT;     (* Transporters[trans].DripTrayDelay  — tenths of second *)
END_VAR

VAR
  vFromIdx                  : INT;
  vToIdx                    : INT;
END_VAR

STC_FC_CalcTransferTime := 0.0;
IF iFromStn > 0 AND iFromStn <> iToStn THEN
  vFromIdx := iFromStn - MIN_STATION_INDEX;
  vToIdx   := iToStn - MIN_STATION_INDEX;
  IF vFromIdx >= 1 AND vFromIdx <= 25 AND vToIdx >= 1 AND vToIdx <= 25 THEN
    STC_FC_CalcTransferTime :=
      (* Phase 2: lift + dropping + drip tray *)
      INT_TO_REAL(iMove.LiftTime[vFromIdx]) / 10.0
      + INT_TO_REAL(iFromDroppingX10) / 10.0
      + INT_TO_REAL(iDripTrayDelayX10) / 10.0
      (* Phase 3: horizontal travel *)
      + INT_TO_REAL(iMove.Travel[vFromIdx].ToTime[vToIdx]) / 10.0
      (* Phase 4: sink + drip tray + device delay *)
      + INT_TO_REAL(iMove.SinkTime[vToIdx]) / 10.0
      + INT_TO_REAL(iDripTrayDelayX10) / 10.0
      + INT_TO_REAL(iToDeviceDelayX10) / 10.0;
  END_IF;
END_IF;

END_FUNCTION

(* ---- STC_FC_CollectActiveBatches.st ---- *)
(* ===========================================================================================
 *  STC_FC_CollectActiveBatches — Filter active/waiting batches
 *
 *  Company : Galvatek part of the John Cockerill Group
 *  Author  : Jarmo Piipponen
 *  Created : 25.03.2026
 *
 * -------------------------------------------------------------------------------------------
 *  Returns count of matching batches; fills oList via VAR_OUTPUT.
 *
 *  Mode:
 *  iMode = 0 — active (in-production) batches
 *  iMode = 1 — waiting batches (station 114 lookup)
 *
 *  ------------------------------------------------------------------------------------------
 *
 *  Changes:
 *
 *
 *
 *)

FUNCTION STC_FC_CollectActiveBatches : INT   (* returns count *)

(* Introduction of Variables ----------------------------------------------------------------*)

VAR_INPUT
  iMode                    : INT;    (* 0 = all active, 1 = waiting only *)
END_VAR

VAR_EXTERNAL CONSTANT
    MAX_UNITS               : INT;
    MAX_STATION_INDEX        : INT;
    USED                    : INT;
    TO_NONE                 : INT;
    NOT_PROCESSED           : INT;
    IN_PROCESS              : INT;
END_VAR

VAR_EXTERNAL
  Batch                   : ARRAY[1..MAX_UNITS] OF UDT_BatchType;
  Unit                    : ARRAY[1..MAX_UNITS] OF UDT_JC_UnitType;
  TreatmentPrograms                 : ARRAY[1..MAX_UNITS] OF UDT_TreatmentProgramType;
  StationOccupancy             : ARRAY[1..MAX_STATION_INDEX] OF UDT_JC_UnitAtStationType;
END_VAR

VAR_OUTPUT
  oList                    : ARRAY[1..MAX_UNITS] OF INT;  (* unit indices *)
END_VAR

VAR
  vUi                        : INT;
  vCnt                       : INT;
END_VAR

vCnt := 0;
FOR vUi := 1 TO MAX_UNITS DO
  oList[vUi] := 0;
END_FOR;

IF iMode = 1 THEN
  (* ── Waiting batch: direct lookup at station 114 ── *)
  vUi := StationOccupancy[114].UnitId;
  IF vUi >= 1 AND vUi <= MAX_UNITS THEN
    IF Unit[vUi].Status = USED
       AND Unit[vUi].Target = TO_NONE
       AND Batch[vUi].State = NOT_PROCESSED
       AND Batch[vUi].ProgId = TreatmentPrograms[vUi].ProgramId
       AND TreatmentPrograms[vUi].ProgramId > 0 THEN
      vCnt := 1;
      oList[1] := vUi;
    END_IF;
  END_IF;
  STC_FC_CollectActiveBatches := vCnt;
  RETURN;
END_IF;

(* ── Mode 0: active batches — loop ── *)
FOR vUi := 1 TO MAX_UNITS DO
  IF Unit[vUi].Status = USED
     AND Unit[vUi].Target = TO_NONE
     AND Batch[vUi].ProgId = TreatmentPrograms[vUi].ProgramId
     AND TreatmentPrograms[vUi].ProgramId > 0 THEN

    IF Batch[vUi].State = IN_PROCESS
       AND Batch[vUi].CurStage >= 0
       AND Batch[vUi].CurStage <= 99 THEN
      vCnt := vCnt + 1;
      oList[vCnt] := vUi;
    END_IF;
  END_IF;
END_FOR;

STC_FC_CollectActiveBatches := vCnt;

END_FUNCTION

(* ---- STC_FC_CreateTasks.st ---- *)
(* ===========================================================================================
 *  STC_FC_CreateTasks — Build task list from schedule for one unit
 *
 *  Company : Galvatek part of the John Cockerill Group
 *  Author  : Jarmo Piipponen
 *  Created : 25.03.2026
 *
 * -------------------------------------------------------------------------------------------
 *  Shared FC: both TSK and DEP call this with different arrays.
 *  Creates transporter tasks from the calculated schedule stages
 *  and appends them to the task queues.
 *
 *  ------------------------------------------------------------------------------------------
 *
 *  Changes:
 *
 *
 *
 *)

FUNCTION STC_FC_CreateTasks : BOOL

(* Introduction of Variables ----------------------------------------------------------------*)

VAR_INPUT
  iUnit                    : INT;
END_VAR

VAR_IN_OUT  (* array sizes must match GVL_JC_Constants: 10=MAX_UNITS, 3=MAX_TRANSPORTERS *)
  ioSchedule               : ARRAY[1..10] OF UDT_JC_TskScheduleType;
  ioTask                   : ARRAY[1..3] OF UDT_JC_TskQueueType;
END_VAR

VAR_EXTERNAL CONSTANT
    MAX_TRANSPORTERS        : INT;
    MAX_UNITS               : INT;
    MAX_TASK_QUEUE          : INT;
    MIN_STATION_INDEX        : INT;
    MAX_STATION_INDEX        : INT;
END_VAR

VAR_EXTERNAL
  Transporters                     : ARRAY[0..MAX_TRANSPORTERS] OF UDT_TransporterType;
  Stations                 : ARRAY[MIN_STATION_INDEX..MAX_STATION_INDEX] OF UDT_StationType;
END_VAR

VAR
  vSi                        : INT;
  vSc                        : INT;
  vLiftStn                  : INT;
  vSinkStn                  : INT;
  vTid                       : INT;
  vQi                        : INT;
  vFB_Find                   : STC_FB_FindTransporter;
  vEffLiftStn              : INT;
END_VAR

STC_FC_CreateTasks := FALSE;
IF iUnit < 1 OR iUnit > MAX_UNITS THEN RETURN; END_IF;

vSc := ioSchedule[iUnit].StageCount;
IF vSc < 1 THEN RETURN; END_IF;

(* Start from 0 if Stages[0] exists (prepend), else from 1 *)
FOR vSi := 0 TO vSc - 1 DO
  IF ioSchedule[iUnit].Stages[vSi].station = 0 THEN
    (* Skip unused stage slot *)
  ELSE
    vLiftStn := ioSchedule[iUnit].Stages[vSi].station;
    vSinkStn := ioSchedule[iUnit].Stages[vSi + 1].station;

    IF vLiftStn > 0 AND vSinkStn > 0 THEN
      vEffLiftStn := vLiftStn;
      IF vLiftStn >= MIN_STATION_INDEX AND vLiftStn <= MAX_STATION_INDEX
         AND vSinkStn >= MIN_STATION_INDEX AND vSinkStn <= MAX_STATION_INDEX THEN
        IF Stations[vLiftStn].Crosstransport > 0
           AND Stations[vLiftStn].ChangeStation > 0
           AND Stations[vLiftStn].YPosition <> Stations[vSinkStn].YPosition THEN
          vEffLiftStn := Stations[vLiftStn].ChangeStation;
        END_IF;
      END_IF;

      vFB_Find(iLiftStn := vEffLiftStn, iSinkStn := vSinkStn);
      vTid := vFB_Find.oTrans;

      IF vTid >= 1 AND vTid <= 3 THEN
        vQi := ioTask[vTid].Count + 1;
        IF vQi <= MAX_TASK_QUEUE THEN
          ioTask[vTid].Queue[vQi].Unit         := iUnit;
          ioTask[vTid].Queue[vQi].Stage        := ioSchedule[iUnit].Stages[vSi + 1].ProgramStage;
          ioTask[vTid].Queue[vQi].SrcStage     := ioSchedule[iUnit].Stages[vSi].ProgramStage;
          ioTask[vTid].Queue[vQi].LiftStationTarget := vEffLiftStn;
          ioTask[vTid].Queue[vQi].SinkStationTarget := vSinkStn;
          ioTask[vTid].Queue[vQi].StartTime   := ioSchedule[iUnit].Stages[vSi].ExitTime;
          ioTask[vTid].Queue[vQi].FinishTime  := ioSchedule[iUnit].Stages[vSi + 1].EntryTime;
          ioTask[vTid].Queue[vQi].CalcTime    := ioSchedule[iUnit].Stages[vSi].CalcTime;
          ioTask[vTid].Queue[vQi].MinTime     := ioSchedule[iUnit].Stages[vSi].MinTime;
          ioTask[vTid].Queue[vQi].MaxTime     := ioSchedule[iUnit].Stages[vSi].MaxTime;
          ioTask[vTid].Count := vQi;
        END_IF;
      END_IF;
    END_IF;
  END_IF; (* skip unused stage slot *)
END_FOR;

STC_FC_CreateTasks := TRUE;

END_FUNCTION
